Fanuc KAREL source: kt00372.KL

-- PROVISIONAL review KL for V770-1; original PC SHA256 b805c99445981cec714856c5b019887158fdcf01ea983b84cd6f394af0e5e038
-- Incomplete behavior may be omitted. Consult companion uncertainty JSON. Do not deploy.
PROGRAM KT00372
%NOLOCKGROUP
VAR
  R1 : REAL
  OUT : BOOLEAN
-- UNRESOLVED_DECL H2 type=002017
BEGIN
  -- UNRESOLVED_PC offsets 5-16; opcodes 2E,23
  -- UNRESOLVED_PC offsets 21-35; opcodes 2E,22,9D,33,B4
  -- UNRESOLVED_PC offsets 40-63; opcodes 21,22,9D,33,B3,64,70,23
  -- UNRESOLVED_PC offsets 68-72; opcodes 7F
END KT00372
